// Mitsubishi GX Works2 project: Termin3_Prvi_zadatak   PLC: FX3S

// task Task_01 (event TRUE, interval 0, priority 31): POU_01

PROGRAM POU_01
VAR
  START : BOOL;
  STOPS : BOOL;
  ukljuceno : BOOL;
  TON_1 : TON;
  vreme1 : TIME;
  Tizl1 : BOOL;
  CTU_1 : CTU;
  brojac1 : INT;
  izlaz_PLC : BOOL;
  CTU_2 : CTU;
END_VAR
(* structured ladder/FBD written out as ST: instructions are called as NAME(EN, inputs, outputs); _pN, _eN, _tN stand for wires *)
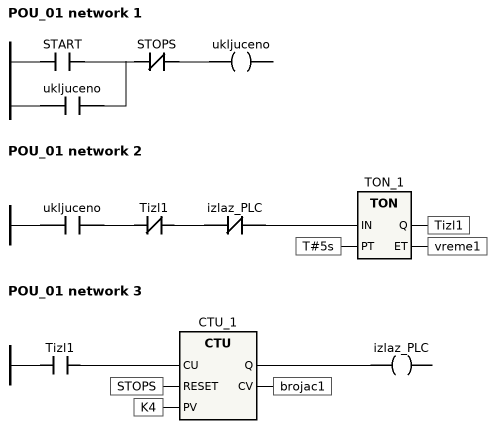
(* network 1 *)
ukljuceno := (START OR ukljuceno) AND NOT STOPS;
(* network 2 *)
TON_1(IN := ukljuceno AND NOT Tizl1 AND NOT izlaz_PLC, PT := T#5s, Q => Tizl1, ET => vreme1);
(* network 3 *)
CTU_1(CU := Tizl1, RESET := STOPS, PV := K4, CV => brojac1);
izlaz_PLC := CTU_1.Q;
END_PROGRAM
